Fanuc KAREL source: kt00262.KL

-- PROVISIONAL review KL for V1013-1; original PC SHA256 33a796fb83048b6e20488811628ec017abcb202a311bcbc2224d77f1984ef4d1
-- Incomplete behavior may be omitted. Consult companion uncertainty JSON. Do not deploy.
PROGRAM KT00262
%NOLOCKGROUP
VAR
  R1 : REAL
  R2 : REAL
  OUT : BOOLEAN
BEGIN
  -- UNRESOLVED_PC offsets 5-16; opcodes 2E,23
  -- UNRESOLVED_PC offsets 21-32; opcodes 2E,23
  -- UNRESOLVED_PC offsets 37-48; opcodes 2E,23
  -- UNRESOLVED_PC offsets 53-64; opcodes 2E,23
  -- UNRESOLVED_PC offsets 69-88; opcodes 21,21,6D,23
  -- UNRESOLVED_PC offsets 93-97; opcodes 7F
END KT00262
